(*

short summary
=============

.. <legal notes>

legal notes
=================
| SPDX-FileCopyrightText: © 2023 ekvip automation GmbH <info@ekvip.de>
| SPDX-License-Identifier: Apache-2.0
| For details check: Apache-2.0_

.. _Apache-2.0: https://www.apache.org/licenses/LICENSE-2.0

.. </legal notes>

methods and properties
======================

*)


FUNCTION_BLOCK AssertionTester EXTENDS CNM_AbstractObject.Object IMPLEMENTS IAttachAssertorContainer
VAR	
	pointerTests 			:PointerAssertionsTests(classToBeTested := 0);
	uxintAssertions			:UxintAssertionTests(classToBeTested := 0);
	usintAssertions			:UsintAssertionTests(classToBeTested := 0);
	uintAssertions			:UintAssertionTests(classToBeTested := 0);
	udintAssertions			:UdintAssertionTests(classToBeTested := 0);
	ulintAssertions			:UlintAssertionTests(classToBeTested := 0);	
	xintAssertions			:XintAssertionTests(classToBeTested := 0);
	sintAssertions			:SintAssertionTests(classToBeTested := 0);
	intAssertions			:IntAssertionTests(classToBeTested := 0);
	dintAssertions			:DintAssertionTests(classToBeTested := 0);
	lintAssertions			:LintAssertionTests(classToBeTested := 0);
	lrealAssertions		 	:LRealAssertionTests(classToBeTested := 0);
	realAssertions			:RealAssertionTests(classToBeTested := 0);
	bitNumberAssertiosByte	:ByteAssertionTests(classToBeTested := 0);
	bitNumberAssertionsWord :WordAssertionTests(classToBeTested := 0);
	bitNumberAssertionDword	:DWordAssertionTests(classToBeTested := 0);
	bitNumberAssertionLWord :LWordAssertionTests(classToBeTested := 0);
	bitNumberAssertionXWord :XWordAssertionTests(classToBeTested := 0);
	binaryTests				:BinaryAssertionsTests(classToBeTested := 0);
	dateAndTimeAssertions 	:DTAssertionTests(classToBeTested := 0);
	ldateAndTimeAssertions 	:LDTAssertionTests(classToBeTested := 0);
	timeTests				:TimeAssertionsTests(classToBeTested := 0);
	ltimeTests				:LTimeAssertionsTests(classToBeTested := 0);
	windows125xStringTests	:Windows125xStringAssertionTests(classToBeTested := 0);
	unicodeUtf8StringTests	:UnicodeUtf8StringAssertionTests(classToBeTested := 0);
	unicodeUtf16StringTests	:UnicodeUtf16StringAssertionTests(classToBeTested := 0);
	objectTests				:ObjectAssertionsTests(classToBeTested := 0);
	dateAssertions			:DateAssertionTests(classToBeTested := 0);
	ldateAssertions			:LDateAssertionTests(classToBeTested := 0);
	timeOfDayAssertions 	:TODAssertionTests(classToBeTested := 0);
	ltimeOfDayAssertions 	:LTODAssertionTests(classToBeTested := 0);
END_VAR

(*

short summary
=============

.. <legal notes>

legal notes
=================
| SPDX-FileCopyrightText: © 2023 ekvip automation GmbH <info@ekvip.de>
| SPDX-License-Identifier: Apache-2.0
| For details check: Apache-2.0_

.. _Apache-2.0: https://www.apache.org/licenses/LICENSE-2.0

.. </legal notes>

*)

PROPERTY attachAssertorContainer : IAssertorContainer
SET

THIS^.timeTests.attachAssertorContainer					:= attachAssertorContainer;
THIS^.ltimeTests.attachAssertorContainer				:= attachAssertorContainer;
THIS^.windows125xStringTests.attachAssertorContainer	:= attachAssertorContainer;
THIS^.unicodeUtf8StringTests.attachAssertorContainer	:= attachAssertorContainer;
THIS^.unicodeUtf16StringTests.attachAssertorContainer	:= attachAssertorContainer;
THIS^.objectTests.attachAssertorContainer 				:= attachAssertorContainer;
THIS^.pointerTests.attachAssertorContainer 				:= attachAssertorContainer;
THIS^.binaryTests.attachAssertorContainer 				:= attachAssertorContainer;
THIS^.lrealAssertions.attachAssertorContainer 			:= attachAssertorContainer;
THIS^.realAssertions.attachAssertorContainer 			:= attachAssertorContainer;
THIS^.dateAssertions.attachAssertorContainer 			:= attachAssertorContainer;
THIS^.ldateAssertions.attachAssertorContainer 			:= attachAssertorContainer;
THIS^.dateAndTimeAssertions.attachAssertorContainer		:= attachAssertorContainer;
THIS^.ldateAndTimeAssertions.attachAssertorContainer	:= attachAssertorContainer;
THIS^.timeOfDayAssertions.attachAssertorContainer		:= attachAssertorContainer;
THIS^.ltimeOfDayAssertions.attachAssertorContainer		:= attachAssertorContainer;
THIS^.usintAssertions.attachAssertorContainer			:= attachAssertorContainer;
THIS^.uintAssertions.attachAssertorContainer			:= attachAssertorContainer;
THIS^.udintAssertions.attachAssertorContainer			:= attachAssertorContainer;
THIS^.ulintAssertions.attachAssertorContainer			:= attachAssertorContainer;
THIS^.uxintAssertions.attachAssertorContainer			:= attachAssertorContainer;
THIS^.sintAssertions.attachAssertorContainer			:= attachAssertorContainer;
THIS^.intAssertions.attachAssertorContainer				:= attachAssertorContainer;
THIS^.dintAssertions.attachAssertorContainer			:= attachAssertorContainer;
THIS^.lintAssertions.attachAssertorContainer			:= attachAssertorContainer;
THIS^.xintAssertions.attachAssertorContainer			:= attachAssertorContainer;
THIS^.bitNumberAssertiosByte.attachAssertorContainer	:= attachAssertorContainer;
THIS^.bitNumberAssertionsWord.attachAssertorContainer	:= attachAssertorContainer;
THIS^.bitNumberAssertionDword.attachAssertorContainer	:= attachAssertorContainer;
THIS^.bitNumberAssertionLWord.attachAssertorContainer	:= attachAssertorContainer;
THIS^.bitNumberAssertionXWord.attachAssertorContainer	:= attachAssertorContainer;
END_SET
END_PROPERTY

(*

short summary
=============

.. <legal notes>

legal notes
=================
| SPDX-FileCopyrightText: © 2023 ekvip automation GmbH <info@ekvip.de>
| SPDX-License-Identifier: Apache-2.0
| For details check: Apache-2.0_

.. _Apache-2.0: https://www.apache.org/licenses/LICENSE-2.0

.. </legal notes>

*)

PROPERTY className :CNM_AbstractObject.ClassName
GET
(*

short summary
=============

.. <legal notes>

legal notes
=================
| SPDX-FileCopyrightText: © 2023 ekvip automation GmbH <info@ekvip.de>
| SPDX-License-Identifier: Apache-2.0
| For details check: Apache-2.0_

.. _Apache-2.0: https://www.apache.org/licenses/LICENSE-2.0

.. </legal notes>

*)

VAR
END_VAR
className := 'AssertionTester';
END_GET
END_PROPERTY

(*

short summary
=================
The constructor ``FB_init`` is needed to create an unique hash code.
The hash code is a pseudo random number create with a xorshift_ algorithm.
It can be overwritten on derivations, because it will be called implicit, ``SUPER^.FB_init()`` is not required.
For more information check: `Behavoir with derived function blocks`_

.. _Behavoir with derived function blocks: https://infosys.beckhoff.com/content/1033/tc3_plc_intro/5482088715.html?id=6983869892358031022
.. _xorshift: https://en.wikipedia.org/wiki/Xorshift

.. <legal notes>

legal notes
=================
| SPDX-FileCopyrightText: © 2022 ekvip automation GmbH <info@ekvip.de>
| SPDX-License-Identifier: Apache-2.0
| For details check: Apache-2.0_

.. _Apache-2.0: https://www.apache.org/licenses/LICENSE-2.0

.. </legal notes>

parameters
=================

*)

METHOD FB_init :BOOL
VAR_INPUT
	(* if TRUE, the retain variables are initialized (warm start / cold start)*)
	bInitRetains	:BOOL;
	(* if TRUE, the instance afterwards gets moved into the copy code (online change) *)
	bInCopyCode		:BOOL;
	(* assertor class to test *)
	classToBeTested :IAssertorContainer;
END_VAR
VAR
	{attribute 'hide'}
	newHashstate3		:CNM_AbstractObject.Hashcode;
END_VAR
VAR CONSTANT
	{attribute 'hide'}
	NUMBER_OF_LEFT_SHIFTS		:UINT	:= 17;
	{attribute 'hide'}
	NUMBER_OF_LEFT_ROTATIONS	:UINT   := 45;
END_VAR
THIS^.attachAssertorContainer := classToBeTested;
END_METHOD

END_FUNCTION_BLOCK

(* stored: Version 1.1.0.1, ProductVersion 3.1.4026.12
   POU AssertionTester: Id {062a13c0-32f4-400a-837d-0e73b4c206ee}, SpecialFunc None
   Property attachAssertorContainer: Id {b2bc5940-b411-4963-89b7-9f29b7800efd}
   Set Set: Id {e2fd7566-6860-4b16-b058-8285801ebad1}
   Property className: Id {5957afeb-394c-4474-bbac-a3ea99270db1}
   Get Get: Id {6e0df682-d4b6-418d-b9d3-d8540a0dfc49}
   Method FB_init: Id {f7a3097f-bc3d-4201-9704-b6443797c814} *)
